FUNCTION F_RemoveProjectName : STRING(255)
VAR_INPUT
	path	: STRING(255);
END_VAR

///////////////////////////////////////////////////////////////////////////////
// F_RemoveProjectName
//
// v1.0.0
///////////////////////////////////////////////////////////////////////////////

F_RemoveProjectName := DELETE(path, LEN(TwinCAT_SystemInfoVarList._AppInfo.ProjectName) + FIND(path, TwinCAT_SystemInfoVarList._AppInfo.ProjectName), 1);
F_RemoveProjectName := F_ToLCase(F_RemoveProjectName);

END_FUNCTION

(* stored: Version 1.1.0.1, ProductVersion 3.1.4024.10
   POU F_RemoveProjectName: Id {c59f1d5c-137d-4730-a01c-a187e653e51b}, SpecialFunc None *)
